(* CODESYS project CtaSysMotor_1.0.0.0.library
   Description: Motor Library der CTA
   Version: 1.0.0.0
   Title: CtaSysMotor
   Author: SIS
   Company: CTA
   Placeholder: CtaSysMotor
   DocFormat: reStructuredText
   DefaultNamespace: CtaSysMotor
   CompiledLibraryCompatibilityVersion: CODESYS V3.5 SP16 Patch 3
   LanguageModelAttribute: qualified-access-only

Project tree, tasks and I/O mapping:
  libraries: Standard, 3.5.18.0 (System); CtaSysConfig, 1.0.0.2 (CTA); CtaAppTime, 1.0.0.1 (CTA)
  40 Visualizations/
  30 Program Organization Units/
    function block fbMotor [ST]: proGeregelt, proEnHandEin, proHandEin, proHandAus, proAuto, proHandStellwert
    Safety Input/
      function block fbSafetyInput [ST]: proError, proOK
    function block fbOperationDataCounter_old [ST]
    function block fbOperationDataCounter [ST]: proRunTil
  00000000-0000-0000-0000-000000000000|D:\CoDeSys\LibrariesV3\trunk\Intern\CAA\CAA Template\3.4.0.0 draft\Placeholder.xml
  00000000-0000-0000-0000-000000000000|D:\CoDeSys\LibrariesV3\trunk\Intern\CAA\CAA Template\3.2.0.3 draft\Prefix.pdf
  00000000-0000-0000-0000-000000000000|D:\CoDeSys\LibrariesV3\trunk\Intern\CAA\CAA Template\3.5.2.0 draft\Placeholder.xml
  20 Structs/
  50 Images/
  10 Documenation/
    global variables VersionHistory
    global variables readMe
  21 Interface/
  11 Library Parameter/
  12 Konstanten/
  60 Textlisten/
  13 Globale Variablen/
  text list GlobalTextList
*)

// 10 Documenation/VersionHistory
(* 

.. image:: ../../Images/CTA_Logo.jpg
   :align: right
   :width: 15% 

**Vorlage**   


============ =========== =========== ============================================
**Date**     **Version** **Author**  **Change**
------------ ----------- ----------- --------------------------------------------
04.03.2021   0.0.0.0     SIS         Vorlage erstellt

============ =========== =========== ============================================


*)
VAR_GLOBAL
    stInfo : STRING:= '0.0.0.0, Vorlage, CTA';
END_VAR

// 10 Documenation/readMe
(*

**ReadMe**
 
|	**Empfehlung**
|
|	Dokumentrieren Sie die Library für eine nachhaltige Entwicklung
|     
| *Beispiel*
| 
| Dies ist die Vorlage Library der CTA. Erstellen Sie ihre Library anhand dieser Vorlage.
*)

VAR_GLOBAL
    xReadMeDone              :   BOOL;
END_VAR

// 30 Program Organization Units/fbMotor
FUNCTION_BLOCK fbMotor
VAR_INPUT
    xEn                   :   BOOL;
    xFreigabe             :   BOOL;
    rFreigabeY            :   REAL;
    xSafetyStop           :   BOOL;
    fbxEnHandEin          :   REFERENCE TO CtaSysConfig.fbBOOL;
    fbxGeregelt           :   REFERENCE TO CtaSysConfig.fbBOOL;
    fbuiHandMode          :   REFERENCE TO CtaSysConfig.fbUINT;
    fbrStellwertHandY     :   REFERENCE TO CtaSysConfig.fbREAL;     
END_VAR   
VAR_OUTPUT          
    xOn                   :   BOOL;
    rOnY                  :   REAL;
    xHand                 :   BOOL;
END_VAR                   
VAR                       
    SRSTO                 :   SR;           
    _xHandAus             :   BOOL;
    _xHandEin             :   BOOL;
    _xAuto                :   BOOL;
    xVarOk                :   BOOL;
END_VAR

(* Variablen Gültikeit *)
xVarOk := __ISVALIDREF(fbxEnHandEin) AND __ISVALIDREF(fbrStellwertHandY) AND __ISVALIDREF(fbxGeregelt) AND __ISVALIDREF(fbuiHandMode);
IF xVarOk THEN
    (* Betriebsmodus *)
    _xAuto    := fbuiHandMode.proValue = 0;
    _xHandAus := fbuiHandMode.proValue = 1;
    _xHandEin := fbuiHandMode.proValue = 2;
END_IF;
(* Sicherheit und Hand Aus *)
IF NOT xSafetyStop AND NOT SRSTO.Q1 AND NOT _xHandAus AND xEn AND xVarOk THEN       
    (* Auto betrieb *)
    IF _xAuto THEN     
        xOn     := xFreigabe;
        (* Stellwert *)
        IF fbxGeregelt.proValue THEN
            rOnY    := SEL(xOn,0,rFreigabeY);
        ELSE
            rOnY    := SEL(xOn,0,100);
        END_IF;
    (* Hand Ein *)
    ELSIF _xHandEin THEN
        IF fbxEnHandEin.proValue THEN
            xOn     := fbxEnHandEin.proValue;
        ELSE
            xOn     := xFreigabe;     
        END_IF;
            rOnY    := fbrStellwertHandY.proValue;
    END_IF;
ELSE
    xOn     := FALSE;
    rOnY    := 0;
END_IF;
(* Hand Modus *)
xHand := _xHandAus OR _xHandEin;
(* STO *)
SRSTO.SET1 := xSafetyStop;
SRSTO.RESET:= NOT xFreigabe;

PROPERTY proGeregelt : BOOL
GET
IF xVarOk THEN
    proGeregelt := fbxGeregelt.proValue;
END_IF;
END_GET
SET
IF xVarOk THEN
    fbxGeregelt.proValue := proGeregelt;
    IF NOT proGeregelt AND NOT proEnHandEin AND proHandEin THEN
        proHandAus := TRUE;    
	END_IF;
END_IF;
END_SET
END_PROPERTY

PROPERTY proEnHandEin : BOOL
SET
IF xVarOk THEN
    (* Freigabe der Funktion Hand Ein *)
    fbxEnHandEin.proValue := proEnHandEin;
    IF NOT proGeregelt AND NOT proEnHandEin AND proHandEin THEN
        proHandAus := TRUE;    
	END_IF;
END_IF;
END_SET
GET
IF xVarOk THEN
    proEnHandEin := fbxEnHandEin.proValue;
END_IF;
END_GET
END_PROPERTY

PROPERTY proHandEin : BOOL
SET
(* Hand Ein *)
IF xVarOk THEN
    IF proHandEin THEN
        IF proEnHandEin OR proGeregelt THEN
            fbuiHandMode.proValue       := 2;  
        END_IF;  
    END_IF;
END_IF;
END_SET
GET
proHandEin := _xHandEin;
END_GET
END_PROPERTY

PROPERTY proHandAus : BOOL
SET
(* Hand Aus *)
IF proHandAus AND xVarOk THEN
    fbuiHandMode.proValue       := 1;
END_IF;
END_SET
GET
proHandAus := _xHandAus;
END_GET
END_PROPERTY

PROPERTY proAuto : BOOL
SET
(* Hand Auto *)
IF proAuto AND xVarOk THEN
    fbuiHandMode.proValue := 0;
END_IF;
END_SET
GET
proAuto := _xAuto;
END_GET
END_PROPERTY

PROPERTY proHandStellwert : REAL
SET
IF xVarOk THEN
    fbrStellwertHandY.proValue := proHandStellwert; 
END_IF;
END_SET
GET
proHandStellwert := fbrStellwertHandY.proValue;
END_GET
END_PROPERTY

END_FUNCTION_BLOCK

// 30 Program Organization Units/Safety Input/fbSafetyInput
FUNCTION_BLOCK fbSafetyInput
VAR_INPUT
    xSafetyIn           :   BOOL;
    xReferenceIn        :   BOOL;
    fbxEnSafetyInput    :   REFERENCE TO CtaSysConfig.fbBOOL;
    fbtStartTime        :   REFERENCE TO CtaSysConfig.fbTIME;
    fbtRunTime          :   REFERENCE TO CtaSysConfig.fbTIME;
END_VAR
VAR_OUTPUT
    xError              :   BOOL;
	xOk					:	BOOL;
END_VAR
VAR
    TON_Safety          :   TON;
    SR_Safety           :   SR;
END_VAR

IF fbxEnSafetyInput.proValue THEN
    (* Start Erkennung *)
    SR_Safety(  SET1    :=  xSafetyIn,
                RESET   :=  NOT xReferenceIn);
    (* Meldung Error *)
    TON_Safety( IN      :=  NOT xSafetyIn AND xReferenceIn,
                PT      :=  SEL(SR_Safety.Q1,fbtStartTime.proValue,fbtRunTime.proValue),
                Q       =>  xError);           
    
ELSE
    xError  := FALSE;
END_IF;                
(* OK *)          
xOk := NOT xError AND SR_Safety.Q1;

PROPERTY proError : BOOL
GET
proError := xError;
END_GET
END_PROPERTY

PROPERTY proOK : BOOL
GET
proOK :=  xOk;
END_GET
END_PROPERTY

END_FUNCTION_BLOCK

// 30 Program Organization Units/fbOperationDataCounter_old
//*******************************************************************************************************************************************************************************************************************************************//
//  Author:         SIS                                                                           																																			 //
//  Version:        1.0.0.0		                                                                      																																		 //
//  Beschreibung:   Betriebszähler                                                                       																																     //
//                                                                          																										                                                	     //
//                                                                             																						 				                                                		 //
//                                                                             																										                                                	  	 //
//*******************************************************************************************************************************************************************************************************************************************//
FUNCTION_BLOCK fbOperationDataCounter_old
//===========================================================================================================================================================================================================================================//
//  Variabeln Deklaration  Input                                                                  																																			 //
//===========================================================================================================================================================================================================================================//
VAR_INPUT
    xOperating              :   BOOL;           // Operations Input = True Anlage lauft Zähler start
    fbudiOperatingStarts    :   REFERENCE TO CtaSysConfig.fbUDINT;
    fbudiOperatingHours     :   REFERENCE TO CtaSysConfig.fbUDINT;
END_VAR
//===========================================================================================================================================================================================================================================//
//  Variabeln Deklaration                                                                                                                                                                                                                    //
//===========================================================================================================================================================================================================================================//
VAR
    xTimeOverMin            :   BOOL;           // Minutentakter
    xOneMinBetrieb          :   BOOL;           // Minutentakter
    diOperatingStartsTemp   :   DINT;           // Übergabevariabel für IN Out
    diOperatingHoursTemp    :   DINT;           // Übergabevariabel für IN Out  
    TON_RunTimeMin          :   TON;            // Timer
    iOperatingMinTemp       :   INT;            // Betriebsminutenzähler
    xOperatingStart         :   BOOL;           // Operationsstart Detektor
END_VAR

//===========================================================================================================================================================================================================================================//
//  Betriebsstunden zähler                                                                                                                                                                                                                   //
//===========================================================================================================================================================================================================================================//
// Prüfen ist Laufzeit Pumpe = 1Min
IF xTimeOverMin THEN
    xOneMinBetrieb := FALSE;
    IF iOperatingMinTemp <= 58 THEN
        iOperatingMinTemp:= iOperatingMinTemp + 1;
    ELSIF iOperatingMinTemp = 59 THEN                       // Aufgrund der IF abfrage erfolgt das = 59 erst in der 60min 
        iOperatingMinTemp:= 0;
        fbudiOperatingHours.proValue:= fbudiOperatingHours.proValue + 1;
    END_IF;
    xTimeOverMin:= FALSE;
END_IF;    

// Timer 1 Min 
TON_RunTimeMin(PT:=T#1M,
                IN:=xOperating AND xOneMinBetrieb,
                Q=>xTimeOverMin); 
                
// Wenn die Pumpe Läuft Starten des Timers                
IF xOperating THEN
    xOneMinBetrieb := TRUE;
ELSE 
    xOneMinBetrieb := FALSE;
END_IF;

//===========================================================================================================================================================================================================================================//
//  Start Zähler                                                                                                                                                                                                                             //
//===========================================================================================================================================================================================================================================//
IF xOperating AND NOT xOperatingStart THEN 
    fbudiOperatingStarts.proValue:= fbudiOperatingStarts.proValue + 1;
    xOperatingStart:= TRUE;
ELSIF NOT xOperating AND xOperatingStart THEN
    xOperatingStart:= FALSE;
END_IF;

END_FUNCTION_BLOCK

// 30 Program Organization Units/fbOperationDataCounter
FUNCTION_BLOCK fbOperationDataCounter
VAR_INPUT
    xOperating              :   BOOL;           // Operations Input = True Anlage lauft Zähler start
    fbudiOperatingStarts    :   CtaSysConfig.ITF_UDINT;
    fbudiOperatingHours     :   CtaSysConfig.ITF_UDINT;
END_VAR
VAR
	fbRunTil				:	CtaAppTime.fbTimeMeasurement;
	ltLastTime				:	LTIME;
    xOperatingStart         :   BOOL;           // Operationsstart Detektor
	usiMin					:	USINT;
END_VAR

IF __QUERYINTERFACE(fbudiOperatingHours,fbudiOperatingHours) AND __QUERYINTERFACE(fbudiOperatingStarts,fbudiOperatingStarts) THEN
	IF xOperating AND NOT xOperatingStart THEN
		fbRunTil.Start();
		ltLastTime := fbRunTil.Stop();
		fbudiOperatingStarts.proValue	:= fbudiOperatingStarts.proValue + 1;
		xOperatingStart 				:= TRUE;
	ELSIF NOT xOperating THEN
		xOperatingStart := FALSE;
	ELSE
		IF ltLastTime + LTIME#1M < fbRunTil.Stop() THEN 
			ltLastTime	:= fbRunTil.Stop();
			usiMin		:= usiMin + 1;
		END_IF;
		IF usiMin >= 60 THEN 
			fbudiOperatingHours.proValue := fbudiOperatingHours.proValue + 1;
			usiMin :=  0;
		END_IF;		
	END_IF;
END_IF;

PROPERTY proRunTil : LTIME
GET
IF xOperating THEN
	proRunTil := fbRunTil.Stop();
ELSE
	proRunTil := LTIME#0S;
END_IF;
END_GET
END_PROPERTY

END_FUNCTION_BLOCK
